# EPICS autosave request: ADCrayDlApp/Db/ADCrayDl_settings.req
$(P)$(R)ColorMode
$(P)$(R)TriggerMode
$(P)$(R)Bin
$(P)$(R)PedestalNumImages
$(P)$(R)ReadoutMode
$(P)$(R)EnableDetectorQuerying
$(P)$(R)VacuumValve
$(P)$(R)Cooler
$(P)$(R)CCDTempSetpoint
$(P)$(R)CoolerTempSetpoint
file "ADBase_settings.req", P=$(P), R=$(R)
